// LS Electric XG5000 project: 0215 로봇
// PLC LSPLC

PROGRAM NewProgram (task: 스캔 프로그램)

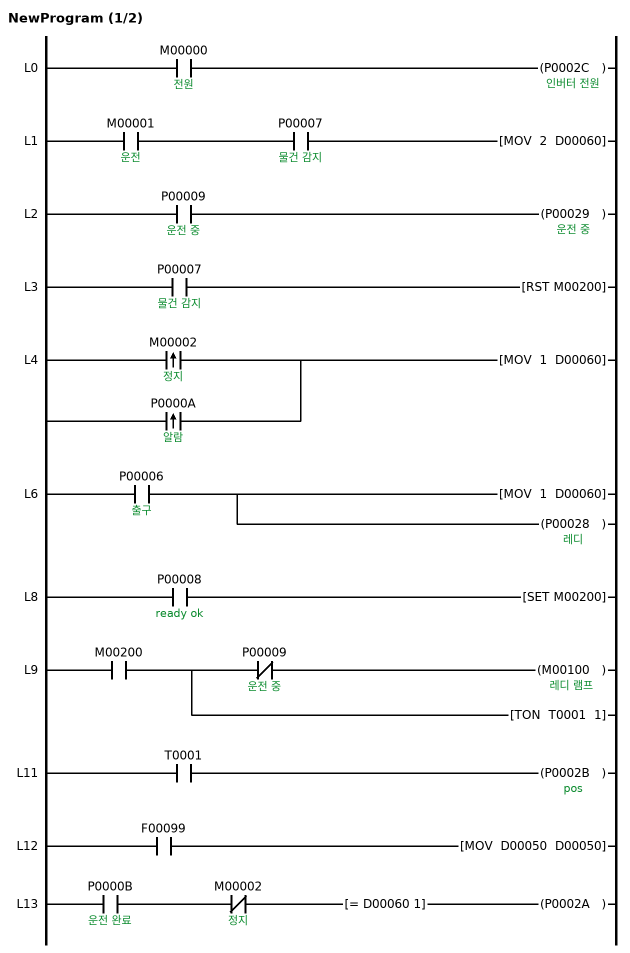
; L0
LOAD      M00000	// 전원
OUT       P0002C	// 인버터 전원
; L1
LOAD      M00001	// 운전
AND       P00007	// 물건 감지
MOV       2 D00060
; L2
LOAD      P00009	// 운전 중
OUT       P00029	// 운전 중
; L3
LOAD      P00007	// 물건 감지
RST       M00200
; L4
LOADP     M00002	// 정지
ORP       P0000A	// 알람
MOV       1 D00060
; L6
LOAD      P00006	// 출구
MOV       1 D00060
OUT       P00028	// 레디
; L8
LOAD      P00008	// ready ok
SET       M00200
; L9
LOAD      M00200
MPUSH
AND NOT   P00009	// 운전 중
OUT       M00100	// 레디 램프
MPOP
TON       T0001 1
; L11
LOAD      T0001
OUT       P0002B	// pos
; L12
LOAD      F00099
MOV       D00050 D00050
; L13
LOAD      P0000B	// 운전 완료
AND NOT   M00002	// 정지
AND=      D00060 1
OUT       P0002A

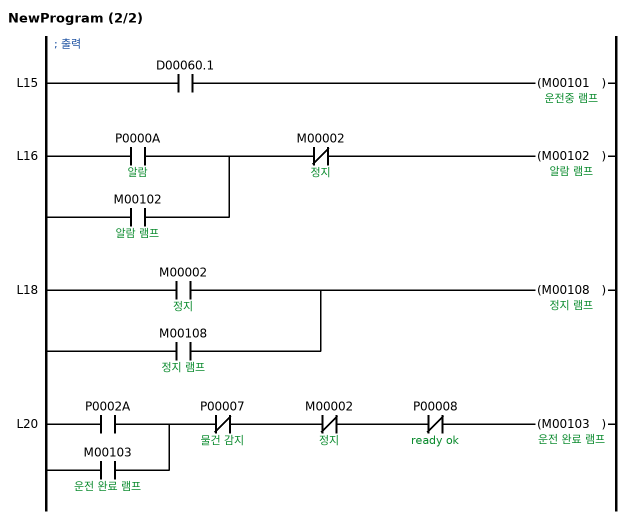
// 출력
; L15
LOAD      D00060.1
OUT       M00101	// 운전중 램프
; L16
LOAD      P0000A	// 알람
OR        M00102	// 알람 램프
AND NOT   M00002	// 정지
OUT       M00102	// 알람 램프
; L18
LOAD      M00002	// 정지
OR        M00108	// 정지 램프
OUT       M00108	// 정지 램프
; L20
LOAD      P0002A
OR        M00103	// 운전 완료 램프
AND NOT   P00007	// 물건 감지
AND NOT   M00002	// 정지
AND NOT   P00008	// ready ok
OUT       M00103	// 운전 완료 램프

VARIABLES AND COMMENTS (devices not used above)
M00004	BIT	포지션 2
M00003	BIT	포지션 1
P00042	BIT	알람 스위치
P00040	BIT	ready ok